PROGRAM PRG_IM1L0_XTES
VAR
	{attribute 'pytmc' := 'pv: IM1L0:XTES'}
	fbIM1L0: FB_XPIM;
	stEL6In: EL6InData22b;
	stEL6Out: EL6OutData22b;
END_VAR

fbIM1L0(
	stYStage := Main.M20,
	stZoomStage := Main.M21,
	stFocusStage := Main.M22,
	stEl6In := stEL6In,
	stEl6Out := stEl6Out,
	fPolished := -87,
	fFrosted := -57,
	fReticle := -27,
	fOut := 0);

END_PROGRAM

(* stored: Version 1.1.0.1, ProductVersion 3.1.4022.12
   POU PRG_IM1L0_XTES: Id {dc3548d0-1688-4ec2-b4ae-fd34a5036e7d}, SpecialFunc None *)
